FUNCTION_BLOCK Test_2
VAR_INPUT
END_VAR
VAR_OUTPUT
END_VAR
VAR
	heyo : REFERENCE TO REAL;
	random: BOOL;
	
END_VAR

random := not random;

PROPERTY PUBLIC P_REAL : REFERENCE TO REAL
SET // PUBLIC
heyo REF= P_REAL;
END_SET
END_PROPERTY

END_FUNCTION_BLOCK

(* stored: Version 1.1.0.1, ProductVersion 3.1.4024.12
   POU Test_2: Id {8d880d00-9f16-4072-8929-a65a8adee6f6}, SpecialFunc None
   Property P_REAL: Id {81ad758e-e003-4e15-8b60-ec7eed54278c}
   Set Set: Id {abd13ffb-a39f-466e-bdb2-f1062c3da2bf} *)
